TEXTLIST AlarmTxtList
  1 = "'AP_PresentSensor'"
  2 = "'AP_PowerOn'"
  3 = "'AP_Ready'"
  4 = "'AP_DeactuatedPLC' "
  5 = "'AP_DeactuatedHwr' "
  6 = "'CellFluidLeakage1' "
  7 = "'CellFluidLeakage2' "
  8 = "'CellGroundFault' "
  9 = "'TesterPresent' "
  10 = "'TesterPowerOn'"
  11 = "'TesterReady' "
  12 = "'TCCellDoorClosed'"
  13 = "'TesterLatchesClosed'"
  14 = "'TIUPresent'"
  15 = ''
  16 = ''
   = ''
END_TEXTLIST

(* stored: Version 1.1.0.1, ProductVersion 3.1.4022.12
   TextList AlarmTxtList: Id {4fd62cf3-b5d6-439e-ac79-2b3642b83901} *)
